{attribute 'GeneratedUsingTerminal: EL3681-0000-0017'}
{attribute addProperty BoxType "EL3681-0000-0017"}
{attribute addProperty Id "UnderrangeBOOL1OverrangeBOOL1Extended_rangeBOOL1Data_InvalidBOOL1Range_InvalidBOOL1Autorange_enabledBOOL1ErrorBOOL1Calibration_in_progressBOOL1TxPDO_StateBOOL1TxPDO_ToggleBOOL1"}
{attribute addProperty CRC "595577615"}
{attribute addProperty Size "10"}
TYPE Status_237FCB0F :
STRUCT
	{attribute addProperty Name "Underrange"}
	Underrange : BOOL;
	{attribute addProperty Name "Overrange"}
	Overrange : BOOL;
	{attribute addProperty Name "Extended_range"}
	Extended_range : BOOL;
	{attribute addProperty Name "Data_Invalid"}
	Data_Invalid : BOOL;
	{attribute addProperty Name "Range_Invalid"}
	Range_Invalid : BOOL;
	{attribute addProperty Name "Autorange_enabled"}
	Autorange_enabled : BOOL;
	{attribute addProperty Name "Error"}
	Error : BOOL;
	{attribute addProperty Name "Calibration_in_progress"}
	Calibration_in_progress : BOOL;
	{attribute addProperty Name "TxPDO_State"}
	TxPDO_State : BOOL;
	{attribute addProperty Name "TxPDO_Toggle"}
	TxPDO_Toggle : BOOL;
END_STRUCT
END_TYPE

(* stored: Version 1.2.0.0, ProductVersion 3.1.4024.9
   DUT Status_237FCB0F: Id {fdec939e-8263-4006-bb30-e177f4820b6c} *)
